(* PLC project cmd_motor_1d1s, GEENSYS ControlBuild 2009-4 (5.10) *)
(* stored: creationDateTime 2009-09-30T16:05:42-01:00 *)

CONFIGURATION cmd_motor_1d1s
  VAR_GLOBAL
    autoMode AT 5 : BOOL := false;
    manualMode AT 6 : BOOL := false;
    autoCmd AT 7 : BOOL := false;
    forwardFB AT 8 : BOOL := false;
    thermalFB AT 9 : BOOL := false;
    forwardPB AT 10 : BOOL := false;
    stopPB AT 11 : BOOL := false;
    acknowledgePB AT 12 : BOOL := false;
    forwardCmd AT 13 : BOOL := false;
    generalFault AT 14 : BOOL := false;
    actions/autoMode AT 5 : BOOL := false;
    actions/manualMode AT 6 : BOOL := false;
    actions/autoCmd AT 7 : BOOL := false;
    actions/forwardPB AT 10 : BOOL := false;
    actions/stopPB AT 11 : BOOL := false;
    actions/generalFault AT 14 : BOOL := false;
    actions/forwardCmd AT 13 : BOOL := false;
    faults/forwardCmd AT 13 : BOOL := false;
    faults/thermalFB AT 9 : BOOL := false;
    faults/forwardFB AT 8 : BOOL := false;
    faults/acknowledgePB AT 12 : BOOL := false;
    faults/generalFault AT 14 : BOOL := false;
    faults/thermalFault AT 15 : BOOL := false;
    faults/forwardFault AT 16 : BOOL := false;
  END_VAR
END_CONFIGURATION
